// TIA Portal project "FB&FC" (V17)

(* hardware
DEVICE "S7-1200 station_1"  S7-1200 Station
   slot 0: "Rack_0"  S7-1200 Rack  Rack  V1.0
   slot 1: "PLC_1"  CPU 1212C DC/DC/DC  6ES7 212-1AE40-0XB0  V4.5
*)

// ===== PLC "PLC_1"  CPU 1212C DC/DC/DC =====

VAR_GLOBAL   // PLC tag table "Default tag table"
   "Start" AT %I0.0 : Bool;
   "Motor" AT %Q0.0 : Bool;
   "Stop" AT %I0.1 : Bool;
   "Fault" AT %I0.2 : Bool;
END_VAR

DATA_BLOCK "Motor_Block_DB"   // DB3
{ S7_Optimized_Access := 'TRUE' }
VERSION : 0.1
// stored: InstanceOfName Motor_Block
"Motor_Block"
BEGIN
END_DATA_BLOCK

FUNCTION_BLOCK "Motor_Block"   // FB1, LAD
{ S7_Optimized_Access := 'TRUE' }
VERSION : 0.1
   VAR_INPUT
      Start : Bool;
      Stop : Bool;
      Fault : Bool;
   END_VAR
   VAR_OUTPUT
      Motor : Bool;
   END_VAR
   VAR
      Latch : Bool;
   END_VAR
BEGIN

REGION Network 1
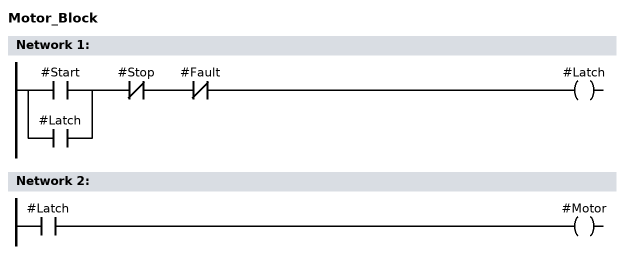
   RUNG wire#powerrail
      Contact( #Start )
      wire#w1
      I_Contact( #Stop )
      I_Contact( #Fault )
      Coil( #Latch )
   END_RUNG
   RUNG wire#powerrail
      Contact( #Latch )
   END_RUNG wire#w1
   // the same network as SCL:
   #Latch := (#Start OR #Latch) AND NOT #Stop AND NOT #Fault;
END_REGION

REGION Network 2
   RUNG wire#powerrail
      Contact( #Latch )
      Coil( #Motor )
   END_RUNG
   // the same network as SCL:
   #Motor := #Latch;
END_REGION
END_FUNCTION_BLOCK

FUNCTION "Motor_SCL" : Void   // FC1, SCL
{ S7_Optimized_Access := 'TRUE' }
VERSION : 0.1
   VAR_INPUT
      Start : Bool;
      Stop : Bool;
      Fault : Bool;
   END_VAR
   VAR_OUTPUT
      Motor : Bool;
   END_VAR
   VAR_TEMP
      latch : Bool;
   END_VAR
BEGIN
   IF #Start AND NOT #Stop AND NOT #Fault THEN
       #latch := TRUE;
   END_IF;
   IF #Stop OR #Fault THEN
       #latch := FALSE;
   END_IF;
   #Motor := #latch;
END_FUNCTION

ORGANIZATION_BLOCK "Main"   // OB1, LAD, ProgramCycle
TITLE = "Main Program Sweep (Cycle)"
{ S7_Optimized_Access := 'TRUE' }
VERSION : 0.1
   VAR_INPUT
      Initial_Call : Bool;   // Initial call of this OB
      Remanence : Bool;   // =True, if remanent data are available
   END_VAR
BEGIN

REGION Network 1
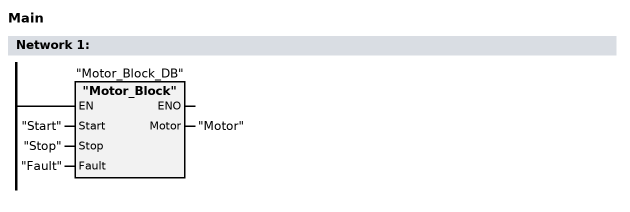
   RUNG wire#powerrail
      "Motor_Block_DB"(Start := "Start", Stop := "Stop", Fault := "Fault", Motor => "Motor")
   END_RUNG
   // the same network as SCL:
   "Motor_Block_DB"(Start := "Start", Stop := "Stop", Fault := "Fault", Motor => "Motor");   // "Motor_Block"
END_REGION
END_ORGANIZATION_BLOCK